FUNCTION_BLOCK FB_FacadeCheck
VAR_INPUT
	nFassade				: INT;
END_VAR
VAR_OUTPUT
	bSunBld_Enable			: BOOL;
	lrFassaden_Orientierung : LREAL;
END_VAR
VAR
END_VAR
// lrFacadeOrientation_Nord

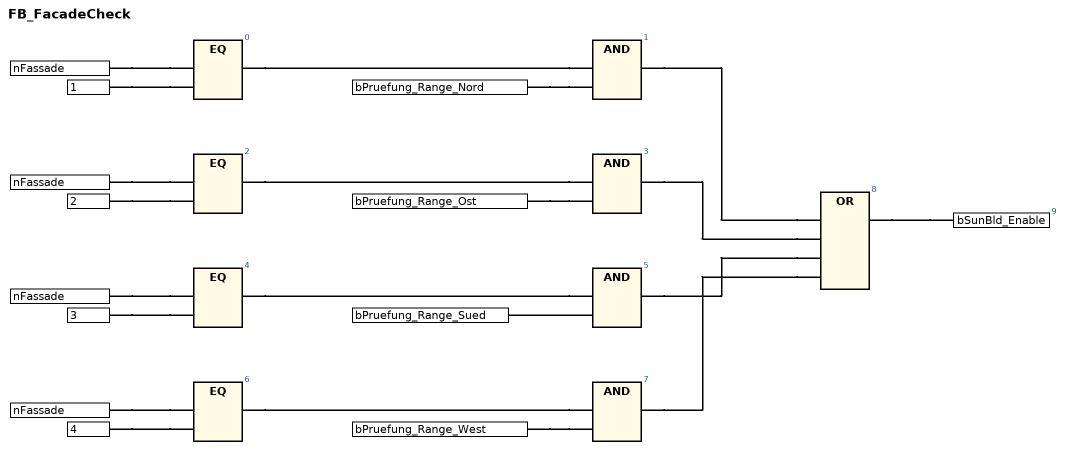
bSunBld_Enable := nFassade = 1 AND bPruefung_Range_Nord OR nFassade = 2 AND bPruefung_Range_Ost OR nFassade = 3 AND bPruefung_Range_Sued OR nFassade = 4 AND bPruefung_Range_West;

END_FUNCTION_BLOCK

(* stored: Version 1.1.0.1, ProductVersion 3.1.4022.7
   POU FB_FacadeCheck: Id {d76910c9-3720-446b-9ef8-89cb0fd3358f}, SpecialFunc None *)
